FUNCTION_BLOCK JackStation
  (* Standard: 61499-2 *)
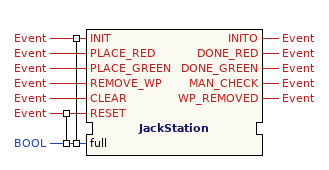
  EVENT_INPUT
    INIT WITH full;
    PLACE_RED;
    PLACE_GREEN;
    REMOVE_WP;
    CLEAR;
    RESET WITH full;
  END_EVENT
  EVENT_OUTPUT
    INITO;
    DONE_RED;
    DONE_GREEN;
    MAN_CHECK;
    WP_REMOVED;
  END_EVENT
  VAR_INPUT
    full : BOOL;
  END_VAR
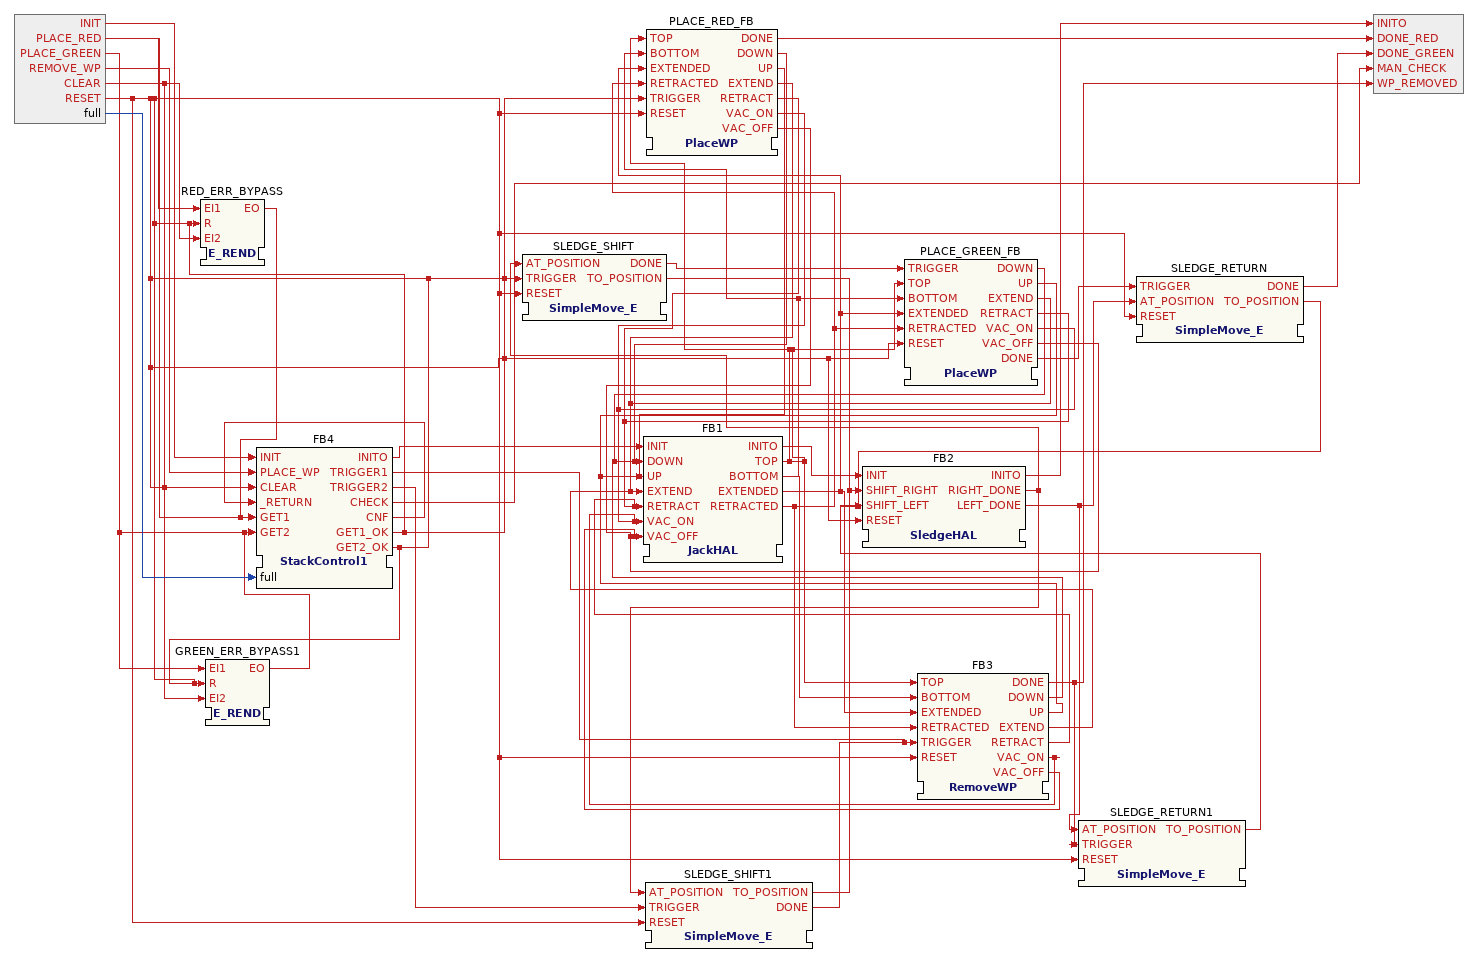
  FBS
    FB1 : JackHAL;
    FB2 : SledgeHAL;
    PLACE_RED_FB : PlaceWP;
    PLACE_GREEN_FB : PlaceWP;
    SLEDGE_SHIFT : SimpleMove_E;
    SLEDGE_RETURN : SimpleMove_E;
    FB3 : RemoveWP;
    SLEDGE_SHIFT1 : SimpleMove_E;
    SLEDGE_RETURN1 : SimpleMove_E;
    FB4 : StackControl1;
    RED_ERR_BYPASS : E_REND;
    GREEN_ERR_BYPASS1 : E_REND;
  END_FBS
  EVENT_CONNECTIONS
    FB4.INITO TO FB1.INIT;
    FB1.INITO TO FB2.INIT;
    FB2.INITO TO INITO;
    PLACE_RED_FB.DONE TO DONE_RED;
    PLACE_RED_FB.DOWN TO FB1.DOWN;
    PLACE_RED_FB.UP TO FB1.UP;
    PLACE_RED_FB.EXTEND TO FB1.EXTEND;
    PLACE_RED_FB.RETRACT TO FB1.RETRACT;
    PLACE_RED_FB.VAC_ON TO FB1.VAC_ON;
    PLACE_RED_FB.VAC_OFF TO FB1.VAC_OFF;
    FB1.TOP TO PLACE_RED_FB.TOP;
    FB1.BOTTOM TO PLACE_RED_FB.BOTTOM;
    FB1.EXTENDED TO PLACE_RED_FB.EXTENDED;
    FB1.RETRACTED TO PLACE_RED_FB.RETRACTED;
    SLEDGE_SHIFT.DONE TO PLACE_GREEN_FB.TRIGGER;
    FB1.TOP TO PLACE_GREEN_FB.TOP;
    FB1.BOTTOM TO PLACE_GREEN_FB.BOTTOM;
    FB1.EXTENDED TO PLACE_GREEN_FB.EXTENDED;
    FB1.RETRACTED TO PLACE_GREEN_FB.RETRACTED;
    PLACE_GREEN_FB.DOWN TO FB1.DOWN;
    PLACE_GREEN_FB.UP TO FB1.UP;
    PLACE_GREEN_FB.EXTEND TO FB1.EXTEND;
    PLACE_GREEN_FB.RETRACT TO FB1.RETRACT;
    PLACE_GREEN_FB.VAC_ON TO FB1.VAC_ON;
    PLACE_GREEN_FB.VAC_OFF TO FB1.VAC_OFF;
    SLEDGE_RETURN.DONE TO DONE_GREEN;
    PLACE_GREEN_FB.DONE TO SLEDGE_RETURN.TRIGGER;
    SLEDGE_SHIFT.TO_POSITION TO FB2.SHIFT_RIGHT;
    FB2.RIGHT_DONE TO SLEDGE_SHIFT.AT_POSITION;
    SLEDGE_RETURN.TO_POSITION TO FB2.SHIFT_LEFT;
    FB2.LEFT_DONE TO SLEDGE_RETURN.AT_POSITION;
    FB1.TOP TO FB3.TOP;
    FB1.BOTTOM TO FB3.BOTTOM;
    FB1.EXTENDED TO FB3.EXTENDED;
    FB1.RETRACTED TO FB3.RETRACTED;
    FB3.DONE TO WP_REMOVED;
    FB3.DOWN TO FB1.DOWN;
    FB3.UP TO FB1.UP;
    FB3.EXTEND TO FB1.EXTEND;
    FB3.RETRACT TO FB1.RETRACT;
    FB3.VAC_ON TO FB1.VAC_ON;
    FB3.VAC_OFF TO FB1.VAC_OFF;
    SLEDGE_SHIFT1.TO_POSITION TO FB2.SHIFT_RIGHT;
    FB2.RIGHT_DONE TO SLEDGE_SHIFT1.AT_POSITION;
    SLEDGE_RETURN1.TO_POSITION TO FB2.SHIFT_LEFT;
    FB2.LEFT_DONE TO SLEDGE_RETURN1.AT_POSITION;
    FB3.DONE TO SLEDGE_RETURN1.TRIGGER;
    SLEDGE_SHIFT1.DONE TO FB3.TRIGGER;
    INIT TO FB4.INIT;
    REMOVE_WP TO FB4.PLACE_WP;
    FB4.TRIGGER1 TO FB3.TRIGGER;
    FB4.TRIGGER2 TO SLEDGE_SHIFT1.TRIGGER;
    FB4.CHECK TO MAN_CHECK;
    CLEAR TO FB4.CLEAR;
    FB4.CNF TO FB4._RETURN;
    PLACE_RED TO FB4.GET1;
    PLACE_GREEN TO FB4.GET2;
    FB4.GET1_OK TO PLACE_RED_FB.TRIGGER;
    FB4.GET2_OK TO SLEDGE_SHIFT.TRIGGER;
    PLACE_RED TO RED_ERR_BYPASS.EI1;
    RED_ERR_BYPASS.EO TO FB4.GET1;
    FB4.GET1_OK TO RED_ERR_BYPASS.R;
    CLEAR TO RED_ERR_BYPASS.EI2;
    GREEN_ERR_BYPASS1.EO TO FB4.GET2;
    PLACE_GREEN TO GREEN_ERR_BYPASS1.EI1;
    FB4.GET2_OK TO GREEN_ERR_BYPASS1.R;
    CLEAR TO GREEN_ERR_BYPASS1.EI2;
    RESET TO PLACE_RED_FB.RESET;
    RESET TO FB4.CLEAR;
    RESET TO GREEN_ERR_BYPASS1.R;
    RESET TO RED_ERR_BYPASS.R;
    RESET TO PLACE_GREEN_FB.RESET;
    RESET TO FB3.RESET;
    RESET TO SLEDGE_SHIFT.RESET;
    RESET TO SLEDGE_RETURN.RESET;
    RESET TO SLEDGE_RETURN1.RESET;
    RESET TO SLEDGE_SHIFT1.RESET;
    RESET TO FB2.RESET;
  END_CONNECTIONS
  DATA_CONNECTIONS
    full TO FB4.full;
  END_CONNECTIONS
END_FUNCTION_BLOCK
